PROGRAM SerialControl
VAR
END_VAR

EL6001.serialCommCtrl(
	Mode := SERIALLINEMODE_EL6_22B,
	pComIn := ADR(EL6001.COMin_EL6001_MASTER),
	SizeComIn := SIZEOF(EL6001.COMin_EL6001_MASTER),
	pComOut := ADR(EL6001.COMout_EL6001_MASTER),
	TxBuffer := EL6001.TxBuffer_MASTER,
	RxBuffer := EL6001.RxBuffer_MASTER);

END_PROGRAM

(* stored: Version 1.1.0.1
   POU SerialControl: Id {f75aaac4-215f-4fc6-bfd3-3f9b3d71cb7a}, SpecialFunc None *)
